(* PLC project Blank Project, Blank Blank 1.0 *)
(* stored: creationDateTime 2016-05-18T21:14:07, modificationDateTime 2017-12-02T21:31:46 *)

PROGRAM Cell3
  VAR
    C2_IR AT %IX0.3 : BOOL := true;
    M2_IR AT %IX0.4 : BOOL := true;
    Main AT %IX0.6 : BOOL := true;
    M2_motor AT %QX0.2 : BOOL := true;
    C3_motor AT %QX0.4 : BOOL := true;
  END_VAR
  VAR
    C3_working : BOOL := false;
    IRset : BOOL := false;
    C3_afterM : BOOL := false;
    Step1 : BOOL := false;
    Step2 : BOOL := false;
    Step3 : BOOL := false;
    Pause : BOOL := false;
    Pause0 : BOOL := false;
    Timer_conveyor : TON;
    Timer_machining : TON;
    TON1 : TON;
    TON2 : TON;
    TON3 : TON;
  END_VAR
  VAR
    JadeProg1 AT %IX0.7 : BOOL := true;
    JadeProg2 AT %IX1.1 : BOOL := true;
    JadeProg3 AT %IX1.2 : BOOL := true;
  END_VAR
  VAR
    TON4 : TON;
  END_VAR

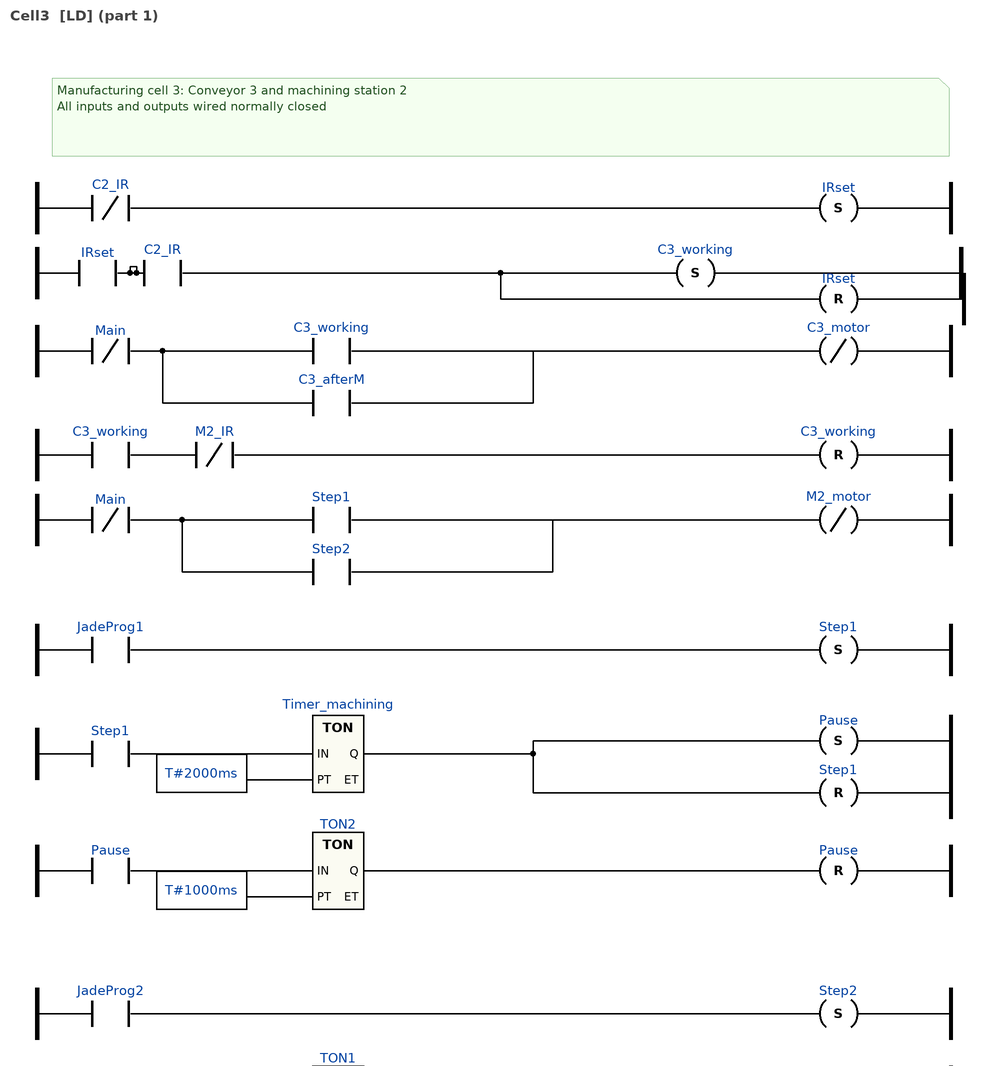
(* LD diagram, written out as Structured Text *)
(* Manufacturing cell 3: Conveyor 3 and machining station 2
All inputs and outputs wired normally closed *)
IF NOT C2_IR THEN IRset := TRUE; END_IF;
IF IRset AND C2_IR THEN C3_working := TRUE; END_IF;
IF IRset AND C2_IR THEN IRset := FALSE; END_IF;
C3_motor := NOT (NOT Main AND (C3_working OR C3_afterM));
IF C3_working AND NOT M2_IR THEN C3_working := FALSE; END_IF;
M2_motor := NOT (NOT Main AND (Step1 OR Step2));
IF JadeProg1 THEN Step1 := TRUE; END_IF;
Timer_machining(IN := Step1, PT := T#2000ms);
IF Timer_machining.Q THEN Pause := TRUE; END_IF;
IF Timer_machining.Q THEN Step1 := FALSE; END_IF;
TON2(IN := Pause, PT := T#1000ms);
IF TON2.Q THEN Pause := FALSE; END_IF;
IF JadeProg2 THEN Step2 := TRUE; END_IF;
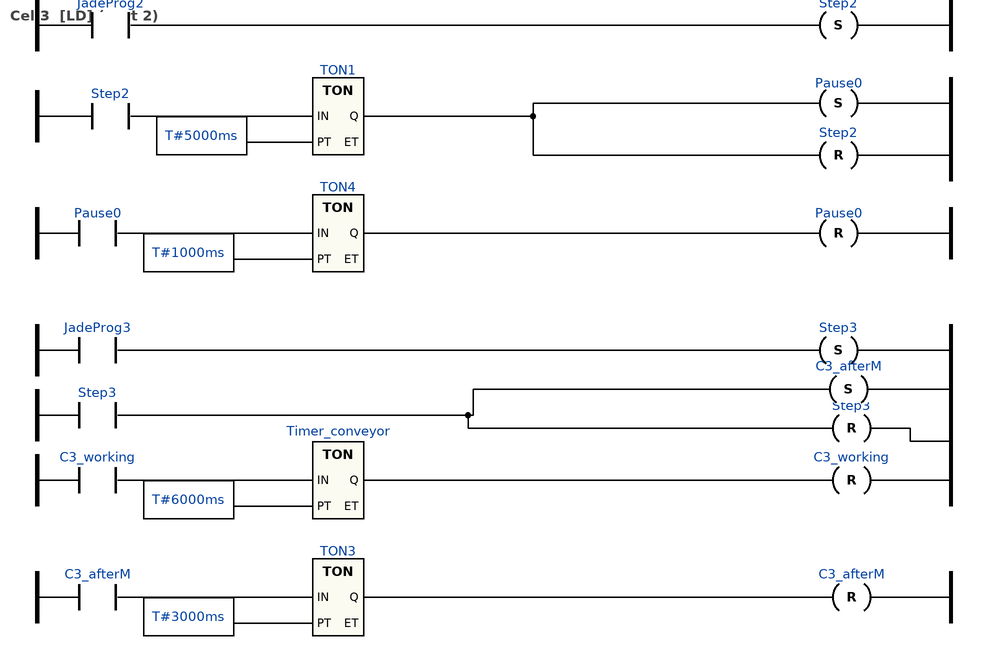
TON1(IN := Step2, PT := T#5000ms);
IF TON1.Q THEN Pause0 := TRUE; END_IF;
IF TON1.Q THEN Step2 := FALSE; END_IF;
TON4(IN := Pause0, PT := T#1000ms);
IF TON4.Q THEN Pause0 := FALSE; END_IF;
IF JadeProg3 THEN Step3 := TRUE; END_IF;
IF Step3 THEN C3_afterM := TRUE; END_IF;
IF Step3 THEN Step3 := FALSE; END_IF;
Timer_conveyor(IN := C3_working, PT := T#6000ms);
IF Timer_conveyor.Q THEN C3_working := FALSE; END_IF;
TON3(IN := C3_afterM, PT := T#3000ms);
IF TON3.Q THEN C3_afterM := FALSE; END_IF;
END_PROGRAM

CONFIGURATION Config0
  RESOURCE Res0 ON PLC
    TASK TaskMain(INTERVAL := T#50ms, PRIORITY := 0);
    PROGRAM Inst0 WITH TaskMain : Cell3;
  END_RESOURCE
END_CONFIGURATION
